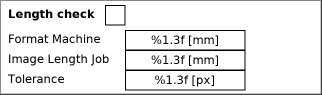
VISUALIZATION _VISU_Pm_Maxliner_ImgLengthCheck  // 322x95
VAR_IN_OUT
	mInst : FB_PrintModule_Maxliner;
END_VAR
    Rectangle (0,0 322x95)
    Rectangle (5,30 120x18), "Format Machine"
    Rectangle (5,5 96x18), "Length check"
    Rectangle (125,30 120x20), "%1.3f [mm]", text variable: mInst._pModuleMachineState^.fSubstrateLen * 1000
    Rectangle (5,50 120x18), "Image Length Job"
    Rectangle (125,50 120x20), "%1.3f [mm]", text variable: mInst.fbWorkerPrint[1]._fCurrentImgDepth * 1000
    RoundedRectangle (105,5 20x20), colour toggle: mInst._pModuleMachineFeedback^.bLengthMismatch
    Rectangle (5,70 120x18), "Tolerance"
    Rectangle (125,70 120x20), "%1.3f [px]", text variable: mInst.fC_FormatLengthTolerance
END_VISUALIZATION

(* stored: Version 1.1.0.1, ProductVersion 3.1.4024.11
   Visu _VISU_Pm_Maxliner_ImgLengthCheck: Id {55ce47de-c618-41d2-ab17-89333c266391} *)
